RoboDK station: Tarea_4_simulacion.rdk

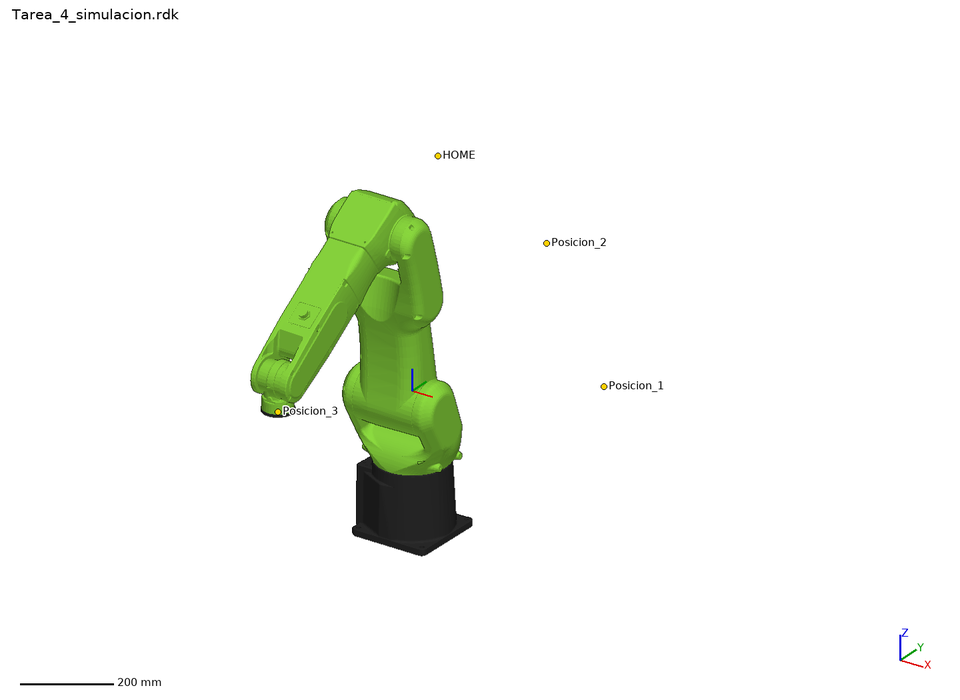
[picture v0: the station drawn from its stored meshes, robots at their saved joint values, targets as dots, program paths as lines]
Station Tarea_4_simulacion (saved by RoboDK 5.8.0). Poses are relative to the parent item; angles as X-Y-Z fixed-axis rotations.
  - frame Fanuc CR-7iA/L Base at (0, 0, 330) mm
    - robot Fanuc CR-7iA/L: 6 axes, payload 7 kg, reach 911 mm, repeatability 0.03 mm, weight 55 kg
        modified DH rows (alpha deg, a mm, theta deg, d mm): 0, 0, 0, 330; -90, 50, -90, 0; 0, 440, 0, 0; -90, 35, 0, 420; 90, 0, 0, 0; -90, 0, 0, 80
        base shift (0, 0, -330) mm
        joint limits [-170, -100, -67, -190, -115, -360] to [170, 145, 213, 190, 115, 360]; home [0, 0, 0, 0, 0, 0]; saved at [-90, 10.532, -33.494, 0, -56.506, 90]
    - target HOME (Cartesian target) at (67.68, 0, 576.29) mm, rotated rx -180 ry -45 rz 0 deg; joints [0, -45, 45, 0, -90, 0] of Fanuc CR-7iA/L
    - target Posicion_1 (Cartesian target) at (500, 0, 150) mm, rotated rx -180 ry 0 rz 0 deg; joints [0, 10.532, -33.494, 0, -56.506, 0] of Fanuc CR-7iA/L
    - target Posicion_2 (Cartesian target) at (0, 500, 150) mm, rotated rx -180 ry 0 rz 0 deg; joints [90, 10.532, -33.494, 0, -56.506, -90] of Fanuc CR-7iA/L
    - target Posicion_3 (Cartesian target) at (0, -500, 150) mm, rotated rx -180 ry 0 rz 0 deg; joints [-90, 10.532, -33.494, 0, -56.506, 90] of Fanuc CR-7iA/L
